{attribute 'linkalways'} 
{attribute 'no_explicit_call' := 'This FB is a CLASS and must be accessed using methods or properties'}
{attribute 'enable_dynamic_creation'}
FUNCTION_BLOCK ABSTRACT AxisCommand EXTENDS Command IMPLEMENTS I_AxisCommand
VAR
	_axisRef : REFERENCE TO Axis;
END_VAR

END_FUNCTION_BLOCK

(* stored: Version 1.1.0.1, ProductVersion 3.1.4024.12
   POU AxisCommand: Id {de57d173-bfb4-446e-800d-5e5d8c6913cd}, SpecialFunc None *)
